TYPE E_DriverOPMode :
(
	DriverOPMode_Pos := 0, // driver position control
	DriverOPMode_Trq :=1, // driver torque control, robot force control
	DriverOPMode_PosTrq :=2, // driver torque control, robot position contorl
	DriverOPMode_Vel :=3, // driver Velocity control
	DriverOPMode_MZPos :=4, //mingzhi driver Position control
	DriverOPMode_cspMZ :=8, //mingzhi driver Sync cycle position mode control
	DriverOPMode_csvMZ :=9 //mingzhi driver Sync cycle position mode control
);
END_TYPE

(* stored: Version 1.1.0.1, ProductVersion 3.1.4024.12
   DUT E_DriverOPMode: Id {a3d3fd7a-69f3-43ec-b98e-ee3226b0a71a} *)
